// TIA Portal V16 export
// export: Created 2022-01-20T18:36:28.9784723Z, ExportSetting WithDefaults, DisplayName Totally Integrated Automation Portal, DisplayVersion V16, DisplayName TIA Portal Version Control Interface, DisplayVersion V16, DisplayName TIA Portal Openness, DisplayVersion V16, DisplayName STEP 7 Professional, DisplayVersion V16, DisplayName STEP 7 Safety, DisplayVersion V16, DisplayName WinCC Advanced, DisplayVersion V16
DATA_BLOCK "DATA"   // DB6
{ S7_Optimized_Access := 'TRUE' }
VERSION : 0.1
// stored: AutoNumber true, IsOnlyStoredInLoadMemory false, IsRetainMemResEnabled false, IsWriteProtectedInAS false, MemoryReserve 100
   VAR
      Receive : Array[0..20] of Char;
      Send : String := 'Hello world!';
      Do_Connect : Bool;
      Passive_Conn_Done : Bool;
   END_VAR
BEGIN
END_DATA_BLOCK
